FUNCTION_BLOCK INTERNAL FB_CoinEjectedState IMPLEMENTS I_State
VAR_INPUT
END_VAR
VAR_OUTPUT
END_VAR
VAR
	pMachine : I_StateMachine;
	customerTakesCoinNext : I_State;
END_VAR

METHOD CustomerTakesCoin : BOOL
ADSLOGSTR(ADSLOG_MSGTYPE_HINT, 'Customer has taken the coin.', '');
pMachine.SetState( customerTakesCoinNext );
END_METHOD

METHOD CustomerTakesProduct : BOOL
END_METHOD

PROPERTY Description : STRING
GET
Description := 'Coin Ejected';
END_GET
END_PROPERTY

METHOD InsertCoin : BOOL
END_METHOD

METHOD PressButton : BOOL
END_METHOD

METHOD SetTransitionStates
VAR_INPUT
	Machine : I_StateMachine;
	CustomerTakesCoinNext : I_State;
END_VAR
THIS^.customerTakesCoinNext := CustomerTakesCoinNext;
THIS^.pMachine := Machine;
END_METHOD

END_FUNCTION_BLOCK

(* stored: Version 1.1.0.1, ProductVersion 3.1.4022.17
   POU FB_CoinEjectedState: Id {65f9b719-bcc3-44e1-96d5-2bce876fa7b7}, SpecialFunc None
   Method CustomerTakesCoin: Id {0bfe65ff-cdb5-477c-9a7f-85028561091f}
   Method CustomerTakesProduct: Id {49b0cba4-d82b-466b-8375-ab02c48a85d5}
   Property Description: Id {1e234bea-11b9-4c49-9972-9acd9825e68d}
   Get Get: Id {905c33c1-31cb-48cb-87d7-b7379a352965}
   Method InsertCoin: Id {812474cc-0340-4650-8083-0f34207c735a}
   Method PressButton: Id {c0931f94-a760-484c-b337-e00a92055645}
   Method SetTransitionStates: Id {ec93e5ef-6b13-4281-bcb7-ce4d6804ee1c} *)
